// Mitsubishi GX Works2 project: final15!!!   PLC: FX3G

// global labels: Global1
VAR_GLOBAL
  StartDay AT X007 : BOOL;
  Oats AT D1111 : REAL;
  Oats_Input AT D1111 : REAL;
  ProteinPowder_Input AT D1114 : REAL;
  Honey_Input AT D1117 : REAL;
  Oats_Amount AT D1113 : REAL;
  ProteinPowder_Amount AT D1116 : REAL;
  Honey_Amount AT D1119 : REAL;
  Exception AT X001 : BOOL;
END_VAR
VAR_GLOBAL CONSTANT
  RequiredClassicOats : REAL := 400;
  RequiredClassicProteinPowder : REAL := 160;
  RequiredClassicHoney : REAL := 120;
END_VAR
VAR_GLOBAL
  MissingMaterialsClassic AT M1 : BOOL;
  Exception1 AT X003 : BOOL;
  MissingMaterials AT M1 : BOOL;
END_VAR
VAR_GLOBAL CONSTANT
  RequiredOats : REAL := 240;
  RequiredProteinPowder : REAL := 160;
  RequiredHoney : REAL := 120;
END_VAR
VAR_GLOBAL
  EmergencyButton AT X005 : BOOL;
  EndDay AT M2 : BOOL;
  MissingMaterialsHold AT M3 : BOOL;
  Y_0 AT Y000 : BOOL;
  Analog_Input_1 AT D8280 : INT;
END_VAR
VAR_GLOBAL CONSTANT
  Div_analog1 : REAL := 400;
  Classic_group : REAL := 5;
END_VAR
VAR_GLOBAL
  Input_1 AT D1121 : REAL;
  Stop_m6 AT M16 : BOOL;
  Snack_Classic AT M6 : BOOL;
END_VAR
VAR_GLOBAL CONSTANT
  Protein_group : REAL := 6;
END_VAR
VAR_GLOBAL
  Snack_Protein AT M7 : BOOL;
  TS_0 AT TS1 : BOOL;
  TS_1 AT TS1 : BOOL;
  Y_3 AT Y003 : BOOL;
  TC_1 AT TC1 : BOOL;
END_VAR
VAR_GLOBAL CONSTANT
  Wait_5_Sec : INT := 50;
  Constant_400 : REAL := 400;
  Constant_160 : REAL := 160;
  Constant_120 : REAL := 120;
END_VAR
VAR_GLOBAL
  Snack_Classic_Stage AT M17 : BOOL;
END_VAR
VAR_GLOBAL CONSTANT
  Constant_240 : REAL := 240;
  Constant_320 : REAL := 320;
END_VAR
VAR_GLOBAL
  Snack_Protein_Stage AT M18 : BOOL;
  Y_1 AT Y001 : BOOL;
  End_Mix AT M20 : BOOL;
  Container_Snack AT D1123 : REAL;
END_VAR
VAR_GLOBAL CONSTANT
  Constant_680 : REAL := 680;
  Constant_720 : REAL := 720;
END_VAR
VAR_GLOBAL
  X_2 AT X002 : BOOL;
  Bake_Snack AT D1125 : REAL;
  Moved_To_Bake AT M21 : BOOL;
  Stop_Blink_After AT M24 : BOOL;
  Monitoring_Bulb AT M22 : BOOL;
  Timer1 AT TC3 : BOOL;
END_VAR
VAR_GLOBAL CONSTANT
  Time1 : INT := 10;
END_VAR
VAR_GLOBAL
  End_Time1 AT TS3 : BOOL;
  Timer2 AT TC4 : BOOL;
END_VAR
VAR_GLOBAL CONSTANT
  Time2 : INT := 10;
END_VAR
VAR_GLOBAL
  End_Time2 AT TS4 : BOOL;
  Y_2 AT Y002 : BOOL;
  Bake_Timer AT TC2 : BOOL;
END_VAR
VAR_GLOBAL CONSTANT
  Bake_4_Sec : INT := 40;
END_VAR
VAR_GLOBAL
  Bake_Timer1 AT TC2 : BOOL;
  Bake_Timer2 AT TC5 : BOOL;
END_VAR
VAR_GLOBAL CONSTANT
  Bake_5_Sec : INT := 50;
END_VAR
VAR_GLOBAL
  TS_2 AT TS1 : BOOL;
  TS_5 AT TS5 : BOOL;
  X_6 AT X006 : BOOL;
  Start_Packing AT M25 : BOOL;
  Package_Counter AT CC2 : BOOL;
  X_0 AT X000 : BOOL;
END_VAR
VAR_GLOBAL CONSTANT
  Package_8 : INT := 8;
END_VAR
VAR_GLOBAL
  Y_4 AT Y004 : BOOL;
  Stop_Y4 AT M26 : BOOL;
  CS_2 AT CS2 : BOOL;
  Package_Container AT D1131 : REAL;
END_VAR
VAR_GLOBAL CONSTANT
  Constant_1 : REAL := 1;
  Div_analog2 : REAL := 40;
END_VAR
VAR_GLOBAL
  output AT D1133 : REAL;
  Analog_Output_1 AT D8282 : INT;
END_VAR

// task Task_01 (event TRUE, interval 0, priority 31): POU_01

PROGRAM POU_01
(* structured ladder/FBD written out as ST: instructions are called as NAME(EN, inputs, outputs); _pN, _eN, _tN stand for wires *)
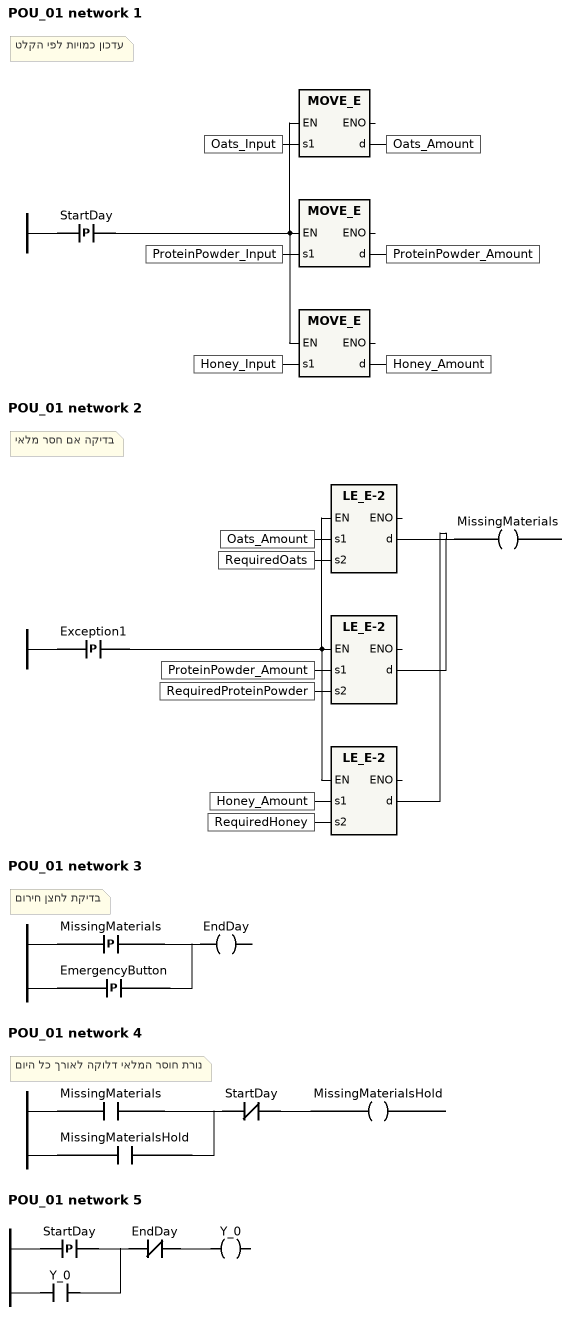
(* network 1 *)
(* עדכון כמויות לפי הקלט *)
_p1 := LDP(TRUE, StartDay);
MOVE_E(_p1, Oats_Input, Oats_Amount);
MOVE_E(_p1, ProteinPowder_Input, ProteinPowder_Amount);
MOVE_E(_p1, Honey_Input, Honey_Amount);
(* network 2 *)
(* בדיקה אם חסר מלאי *)
_p1 := LDP(TRUE, Exception1);
LE_E(_p1, Oats_Amount, RequiredOats, _t2);
LE_E(_p1, ProteinPowder_Amount, RequiredProteinPowder, _t3);
LE_E(_p1, Honey_Amount, RequiredHoney, _t4);
MissingMaterials := _t2 OR _t3 OR _t4;
(* network 3 *)
(* בדיקת לחצן חירום *)
EndDay := LDP(TRUE, MissingMaterials) OR LDP(TRUE, EmergencyButton);
(* network 4 *)
(* נורת חוסר המלאי דלוקה לאורך כל היום *)
MissingMaterialsHold := (MissingMaterials OR MissingMaterialsHold) AND NOT StartDay;
(* network 5 *)
Y_0 := (LDP(TRUE, StartDay) OR Y_0) AND NOT EndDay;
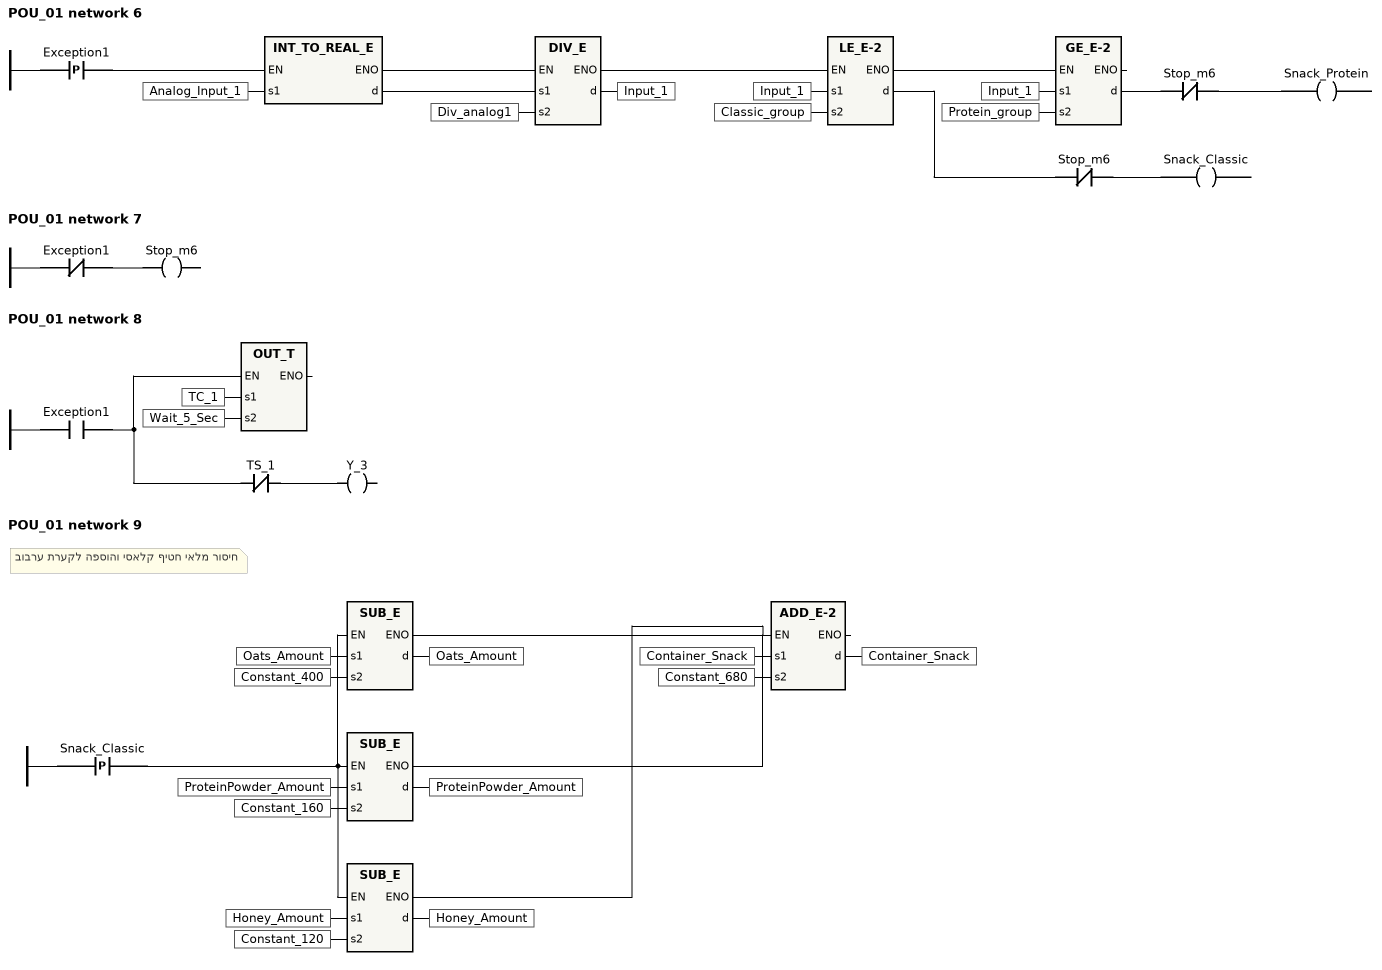
(* network 6 *)
_e2 := INT_TO_REAL_E(LDP(TRUE, Exception1), Analog_Input_1, _t1);
_e3 := DIV_E(_e2, _t1, Div_analog1, Input_1);
_e5 := LE_E(_e3, Input_1, Classic_group, _t4);
GE_E(_e5, Input_1, Protein_group, _t6);
Snack_Protein := _t6 AND NOT Stop_m6;
Snack_Classic := _t4 AND NOT Stop_m6;
(* network 7 *)
Stop_m6 := NOT Exception1;
(* network 8 *)
OUT_T(Exception1, TC_1, Wait_5_Sec);
Y_3 := Exception1 AND NOT TS_1;
(* network 9 *)
(* חיסור מלאי חטיף קלאסי והוספה לקערת ערבוב *)
_p1 := LDP(TRUE, Snack_Classic);
_e2 := SUB_E(_p1, Oats_Amount, Constant_400, Oats_Amount);
_e3 := SUB_E(_p1, ProteinPowder_Amount, Constant_160, ProteinPowder_Amount);
_e4 := SUB_E(_p1, Honey_Amount, Constant_120, Honey_Amount);
ADD_E(_e2 OR _e3 OR _e4, Container_Snack, Constant_680, Container_Snack);
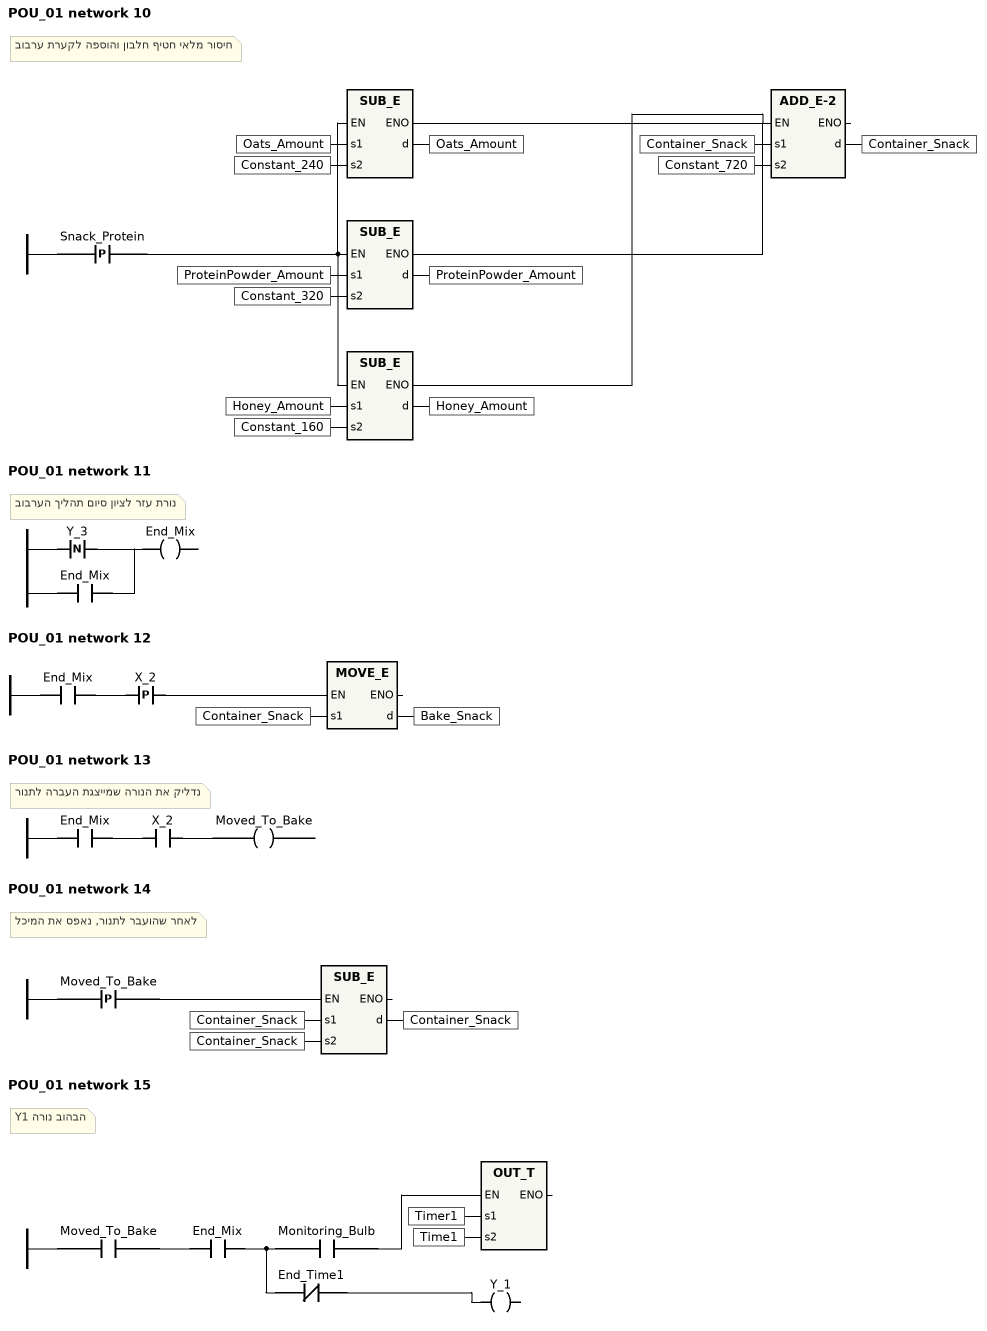
(* network 10 *)
(* חיסור מלאי חטיף חלבון והוספה לקערת ערבוב *)
_p1 := LDP(TRUE, Snack_Protein);
_e2 := SUB_E(_p1, Oats_Amount, Constant_240, Oats_Amount);
_e3 := SUB_E(_p1, ProteinPowder_Amount, Constant_320, ProteinPowder_Amount);
_e4 := SUB_E(_p1, Honey_Amount, Constant_160, Honey_Amount);
ADD_E(_e2 OR _e3 OR _e4, Container_Snack, Constant_720, Container_Snack);
(* network 11 *)
(* נורת עזר לציון סיום תהליך הערבוב *)
End_Mix := LDF(TRUE, Y_3) OR End_Mix;
(* network 12 *)
MOVE_E(End_Mix AND LDP(TRUE, X_2), Container_Snack, Bake_Snack);
(* network 13 *)
(* נדליק את הנורה שמייצגת העברה לתנור *)
Moved_To_Bake := End_Mix AND X_2;
(* network 14 *)
(* לאחר שהועבר לתנור, נאפס את המיכל *)
SUB_E(LDP(TRUE, Moved_To_Bake), Container_Snack, Container_Snack, Container_Snack);
(* network 15 *)
(* הבהוב נורה Y1 *)
_p1 := Moved_To_Bake AND End_Mix;
OUT_T(_p1 AND Monitoring_Bulb, Timer1, Time1);
Y_1 := _p1 AND NOT End_Time1;
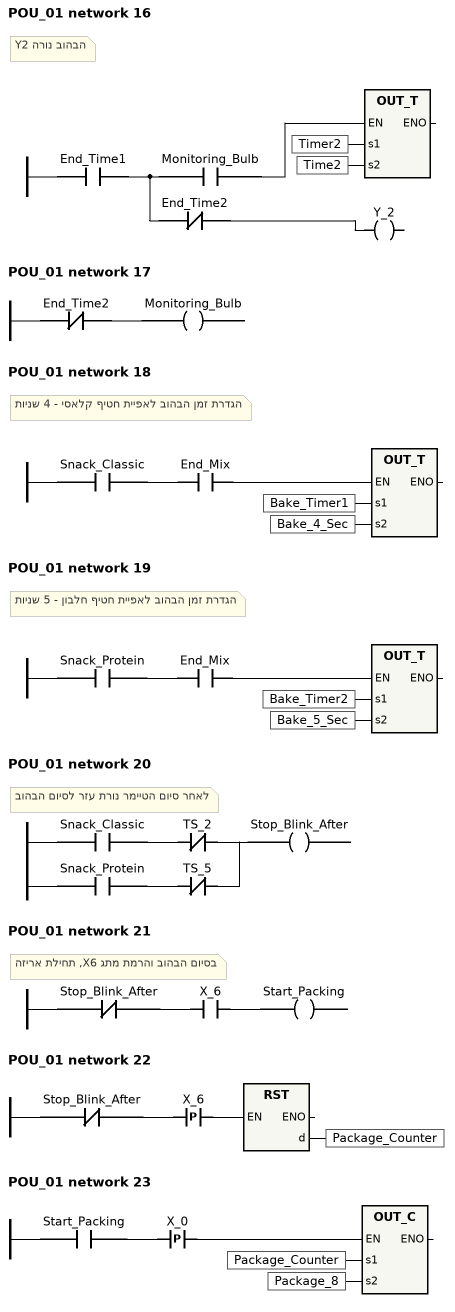
(* network 16 *)
(* הבהוב נורה Y2 *)
OUT_T(End_Time1 AND Monitoring_Bulb, Timer2, Time2);
Y_2 := End_Time1 AND NOT End_Time2;
(* network 17 *)
Monitoring_Bulb := NOT End_Time2;
(* network 18 *)
(* הגדרת זמן הבהוב לאפיית חטיף קלאסי - 4 שניות *)
OUT_T(Snack_Classic AND End_Mix, Bake_Timer1, Bake_4_Sec);
(* network 19 *)
(* הגדרת זמן הבהוב לאפיית חטיף חלבון - 5 שניות *)
OUT_T(Snack_Protein AND End_Mix, Bake_Timer2, Bake_5_Sec);
(* network 20 *)
(* לאחר סיום הטיימר נורת עזר לסיום הבהוב *)
Stop_Blink_After := (Snack_Classic AND NOT TS_2) OR (Snack_Protein AND NOT TS_5);
(* network 21 *)
(* בסיום הבהוב והרמת מתג X6, תחילת אריזה *)
Start_Packing := NOT Stop_Blink_After AND X_6;
(* network 22 *)
RST(NOT Stop_Blink_After AND LDP(TRUE, X_6), Package_Counter);
(* network 23 *)
OUT_C(Start_Packing AND LDP(TRUE, X_0), Package_Counter, Package_8);
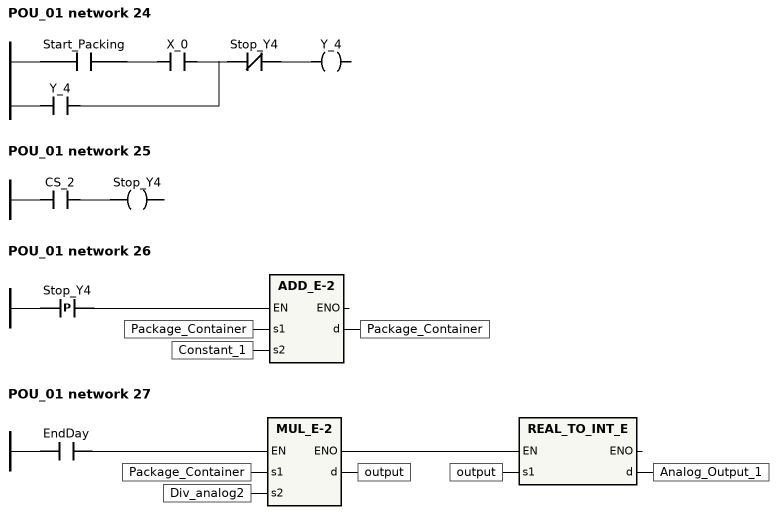
(* network 24 *)
Y_4 := ((Start_Packing AND X_0) OR Y_4) AND NOT Stop_Y4;
(* network 25 *)
Stop_Y4 := CS_2;
(* network 26 *)
ADD_E(LDP(TRUE, Stop_Y4), Package_Container, Constant_1, Package_Container);
(* network 27 *)
_e1 := MUL_E(EndDay, Package_Container, Div_analog2, output);
REAL_TO_INT_E(_e1, output, Analog_Output_1);
END_PROGRAM
